SUBAPPLICATION Uebung_010f4_AX (* SCHLECHTER STIL (Punktabzug!): SoftKey_F1 ODER AuxFunction2_X1 auf DigitalOutput_Q1 mit 2x GreenWhiteBackground statt GreenWhiteBackground3_AX - siehe Uebung_010f3_AX fuer die korrekte Loesung *)
  (* Standard: 61499-2; Description: Copyright (c) 2026 Meisterschulen am Ostbahnhof This program and the accompanying materials are made available under the terms of the Eclipse Public License 2.0 which is available at https://www.eclipse.org/legal/epl-2.0/ SPDX-License-Identifier: EPL-2.0 *)
  (* Version 1.0, 2026-09-06, Franz Höpfinger, Meisterschulen am Ostbahnhof, initial API and implementation and/or initial documentation *)
  PACKAGE Uebungen;
  IMPORT Uebungen::const::UT::DefaultPool::SoftKey_F1;
  IMPORT Uebungen::const::UT::DefaultPool::AuxFunction2_X1;
  IMPORT logiBUS::io::DQ::logiBUS_DO::Output_Q1;
  (* Documentation:
  SCHLECHTER STIL (Punktabzug!) - siehe Uebung_010f3_AX für die korrekte Lösung
   Diese Datei ist absichtlich als Negativbeispiel stehen gelassen: sie erreicht funktional dasselbe wie Uebung_010f3_AX, tut es aber mit unnötig aufgeblähter Verdrahtung.
   Was hier falsch gemacht wurde
    - Statt des dafür gebauten Bausteins GreenWhiteBackground3_AX (nimmt u16ObjId UND u16ObjIdA gleichzeitig und braucht nur einen DI1-Eingang) wurden hier GreenWhiteBackground1_AX und GreenWhiteBackground2_AX als zwei separate Instanzen verdrahtet.
   - Dadurch war fälschlich ein AX_SPLIT_3 (3 Ziele) statt eines simplen AX_SPLIT_2 (2 Ziele) nötig.
   - Die Farbauswahl-Logik (AX_SEL Weiß/Grün) läuft dadurch doppelt statt einmal - unnötiger Ressourcenverbrauch und unnötig große Diagramme, ohne jeden funktionalen Vorteil.
    Lernziel
   Bevor man für einen kombinierten Fall (normales VT-Objekt + Aux-Objekt) mehrere generische Bausteine einzeln zusammenschraubt, erst prüfen, ob es dafür nicht schon einen passenden, fertigen Baustein in der Bibliothek gibt (hier: GreenWhiteBackground3_AX). Vergleichen Sie diese Datei mit Uebung_010f3_AX, um den Unterschied zu sehen.
  *)
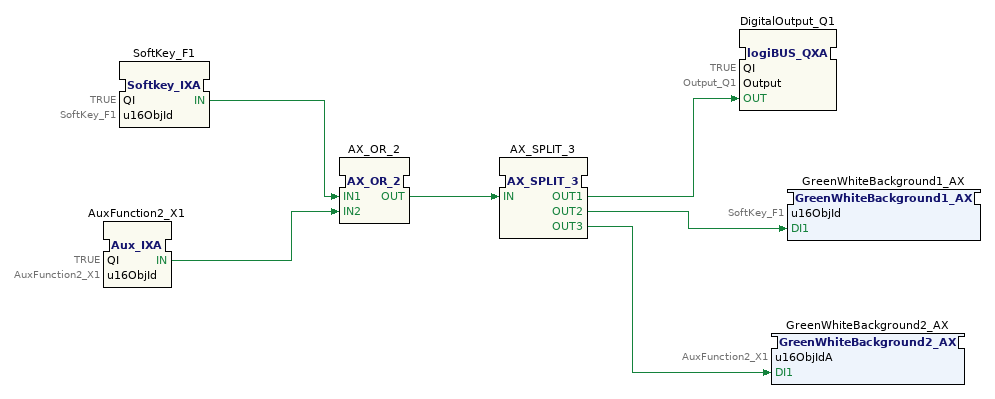
  (* SCHLECHTER STIL - Punktabzug! Hier wurden GreenWhiteBackground1_AX UND GreenWhiteBackground2_AX einzeln verdrahtet (+ AX_SPLIT_3 fuer 3 Ziele), obwohl es mit GreenWhiteBackground3_AX (ein Baustein, u16ObjId + u16ObjIdA, nur AX_SPLIT_2 noetig) genau fuer diesen Fall (1 normales VT-Objekt + 1 Aux-Objekt) schon fertig existiert. Unnoetige Verdopplung der Farbauswahl-Logik (2x AX_SEL statt 1x). Korrekte Loesung: Uebung_010f3_AX. *)
  FBS
    DigitalOutput_Q1 : logiBUS::io::DQ::logiBUS_QXA(QI := TRUE, Output := Output_Q1);
    SoftKey_F1 : isobus::UT::io::Softkey::Softkey_IXA(QI := TRUE, u16ObjId := SoftKey_F1);
    AuxFunction2_X1 : isobus::UT::io::Auxiliary::IN::Aux_IXA(QI := TRUE, u16ObjId := AuxFunction2_X1);
    AX_OR_2 : adapter::booleanOperators::AX_OR_2;
    AX_SPLIT_3 : adapter::events::unidirectional::AX_SPLIT_3;
  END_FBS
  SUBAPPS
    GreenWhiteBackground1_AX : MyLib::sys::GreenWhiteBackground1_AX(u16ObjId := SoftKey_F1);
    GreenWhiteBackground2_AX : MyLib::sys::GreenWhiteBackground2_AX(u16ObjIdA := AuxFunction2_X1);
  END_SUBAPPS
  ADAPTER_CONNECTIONS
    SoftKey_F1.IN TO AX_OR_2.IN1;
    AuxFunction2_X1.IN TO AX_OR_2.IN2;
    AX_OR_2.OUT TO AX_SPLIT_3.IN;
    AX_SPLIT_3.OUT1 TO DigitalOutput_Q1.OUT;
    AX_SPLIT_3.OUT2 TO GreenWhiteBackground1_AX.DI1;
    AX_SPLIT_3.OUT3 TO GreenWhiteBackground2_AX.DI1;
  END_CONNECTIONS
END_SUBAPPLICATION
